TEXTLIST actionSelectList
  0 = 'BRAKE OFF'
  1 = 'BRAKE ON'
  2 = 'DISABLE'
  3 = 'ENABLE'
  4 = 'HOME TO SENSOR'
  5 = 'HOME TO TORQUE'
  6 = 'MOVE TO POSITION'
  7 = 'JOG'
  8 = 'MOVE TO TORQUE'
  9 = 'RESET'
   = ''
END_TEXTLIST

(* stored: Version 1.1.0.1, ProductVersion 3.1.4024.13
   TextList actionSelectList: Id {db282ee1-3f29-4f05-aa01-268fe663affe} *)
